TYPE T_UTC_TIME :
STRUCT
	dcTime:   ULINT;
	mode:     DINT;
END_STRUCT
END_TYPE

(* stored: Version 1.1.0.1, ProductVersion 3.1.4022.9
   DUT T_UTC_TIME: Id {4c9f7993-6638-442a-bc32-de521cf9bd61} *)
